Fanuc KAREL source: kt00535.KL

-- PROVISIONAL review KL for V940-1; original PC SHA256 fd0336ade9c7e2f7f6c337104fe36839b734cdbe18f62ca1d0f35a99f3a1048f
-- Incomplete behavior may be omitted. Consult companion uncertainty JSON. Do not deploy.
PROGRAM KT00535
%NOLOCKGROUP
-- UNRESOLVED_DECL P1 type=000199
-- UNRESOLVED_DECL P2 type=000101
-- UNRESOLVED_DECL OUT type=000102
BEGIN
  -- V9_ZERO_TABLE_METADATA_HINT layout=0001; no indexed target words; source/name/runtime held
  -- UNRESOLVED_PC offsets 5-39; opcodes 49,7E,49,60,7E,4A
  -- UNRESOLVED_PC offsets 44-48; opcodes 7F
END KT00535
